# EPICS autosave request: softGlueApp/Db/DnCntr_settings.req
$(P)$(H)DnCntr-$(N)_CLOCK_Signal
$(P)$(H)DnCntr-$(N)_ENABLE_Signal
$(P)$(H)DnCntr-$(N)_LOAD_Signal
$(P)$(H)DnCntr-$(N)_OUT_Signal
$(P)$(H)DnCntr-$(N)_PRESET
